// TIA Portal V16 export
// export: Created 2024-12-03T15:41:42.3875884Z, ExportSetting WithDefaults, DisplayName Totally Integrated Automation Portal, DisplayVersion V16 Update 6, DisplayName TIA Portal Version Control Interface, DisplayVersion V16 Update 2, DisplayName TIA Portal Openness, DisplayVersion V16 Update 6, DisplayName TIA Portal Teamcenter Gateway, DisplayVersion V16, DisplayName SINAMICS Startdrive Advanced, DisplayVersion V16 Update 5, DisplayName SINAMICS Startdrive G130, G150, S120, S150, SINAMICS MV, S210, DisplayVersion V16 Update 5, DisplayName SINAMICS Startdrive G110M, G120, G120C, G120D, G120P, G115D, DisplayVersion V16 Update 5, DisplayName STEP 7 Professional, DisplayVersion V16 Update 6, DisplayName STEP 7 Safety, DisplayVersion V16, DisplayName WinCC Advanced / Unified PC, DisplayVersion V16 Update 6
FUNCTION_BLOCK "LC_Cognex_DataMan_FB"   // FB15, SCL
{ S7_Optimized_Access := 'TRUE' }
VERSION : 0.1
// stored: AutoNumber true, IsIECCheckEnabled false, IsRetainMemResEnabled false, MemoryReserve 100, SetENOAutomatically false, UDAEnableTagReadback false
   VAR_OUTPUT
      O_Tracking : "Tracking_Simple_UDT_1";
      O_NewResult : Bool;
   END_VAR
   VAR_IN_OUT
      IO_BarcodeScanner : "COGNEX_DATAMAN_LOGIC_UDT";
      IO_UpstreamConv : "Conveyor_UDT";
      IO_CurrentStream : "Conveyor_UDT";
   END_VAR
   VAR
      measureBoxTimer : TONR_TIME;
      scanTimer { S7_SetPoint := 'True'} : TONR_TIME;
      boxLength { S7_SetPoint := 'True'} : Time;
      stepNumber : DInt;
      Step_10_WaitForTrigger : "StepperController";
      Step_20_OnDelay { S7_SetPoint := 'True'} : "StepperController";
      Step_30_Scan { S7_SetPoint := 'True'} : "StepperController";
      Step_40_ParseResult { S7_SetPoint := 'True'} : "StepperController";
      Step_50_ParcelsToClose { S7_SetPoint := 'True'} : "StepperController";
   END_VAR
   VAR_TEMP
      T_Condition : Bool;
      T_Dummy : Bool;
   END_VAR
BEGIN
   REGION #init

       IF #stepNumber = 0 THEN
           #stepNumber := 10;
       END_IF;

   END_REGION

   REGION Measure box

       #measureBoxTimer(IN := #IO_UpstreamConv.Input.SensorAtEndLogic.State
                        AND #IO_UpstreamConv.Input.Running_FB,
                        PT := T#10s);

       IF #IO_UpstreamConv.Input.SensorAtEndLogic.State THEN
           #boxLength := #measureBoxTimer.ET;
           PRESET_TIMER(PT:= #boxLength + #IO_BarcodeScanner.Settings.OffDelay, "TIMER" := #scanTimer);
       END_IF;

       IF NOT #IO_UpstreamConv.Input.SensorAtEndLogic.State THEN
           RESET_TIMER(#measureBoxTimer);
       END_IF;

   END_REGION

   REGION STEP  10: Standby wait FOR trigger

       #T_Condition :=
       #IO_UpstreamConv.Input.SensorAtEndLogic.State
       AND #IO_UpstreamConv.Input.Running_FB
       AND #IO_UpstreamConv.Cmd.ReadyToSent
       AND #IO_CurrentStream.Cmd.ReadyToReceive;

       #Step_10_WaitForTrigger(I_StepNumber := 10,
                               I_NextStepNumber := 20,
                               I_ErrorStepNumber := 50,
                               I_Condition := #T_Condition AND #IO_BarcodeScanner.Status.ReadyForNewScan,
                               I_ErrorConditon := #T_Condition AND NOT #IO_BarcodeScanner.Status.ReadyForNewScan,
                               I_ConditionTIme := T#0ms,
                               I_IgnoreTimeOut := TRUE,
                               IO_StepNumber := #stepNumber);

       IF #Step_10_WaitForTrigger.O_ConditionTrans
           OR #Step_10_WaitForTrigger.O_ErrorTrans THEN
           #IO_BarcodeScanner.Tracking.ID := #IO_UpstreamConv.TrackingStat.Current.ID;
       END_IF;

   END_REGION

   REGION STEP 20: Start trigger command on delay

       #T_Condition := TRUE;

       #Step_20_OnDelay(I_StepNumber := 20,
                               I_NextStepNumber := 30,
                               I_Condition := #T_Condition,
                               I_ConditionTIme := #IO_BarcodeScanner.Settings.OnDelay,
                               I_PauseTimeOut := NOT #IO_CurrentStream.Input.Running_FB,
                               I_AccumulateConditionTIme := TRUE,
                               I_IgnoreTimeOut := TRUE,
                               IO_StepNumber := #stepNumber);

   END_REGION

   REGION STEP 30: TRIGGER MEASURE TIME + OFF DELAY

       //Timer must be external
       #scanTimer(IN:=#stepNumber = 30 AND ( #IO_CurrentStream.Input.Running_FB OR #IO_CurrentStream.Input.SensorAtEndLogic.State),
                  R:=#stepNumber <> 30,
                  Q=> #T_Dummy,
                  PT:=#boxLength);

       #T_Condition := #scanTimer.Q;

       #Step_30_Scan(I_StepNumber := 30,
                               I_NextStepNumber := 40,
                               I_Condition := #T_Condition,
                               I_ConditionTIme := T#0ms,
                               I_IgnoreTimeOut := TRUE,
                               IO_StepNumber := #stepNumber);

   END_REGION

   REGION STEP40: Wait for result

       #Step_40_ParseResult(I_StepNumber:=40,
                            I_NextStepNumber:=10,
                            I_TimeOutStepNumber:=10,
                            I_ConditionTIme := t#0s,
                            I_Condition:=#IO_BarcodeScanner.ReadingResult.NewResult_Pulse,
                            I_TimeOutTime:=#IO_BarcodeScanner.Settings.TimeOut,
                            IO_StepNumber:=#stepNumber);

       IF #IO_BarcodeScanner.ReadingResult.NewResult_Pulse THEN
           "Test_DB".Counter += 1;
       END_IF;

   END_REGION

   REGION STPEP 50: Parcels to close

       #Step_50_ParcelsToClose(I_StepNumber := 50,
                            I_NextStepNumber := 10,
                            I_TimeOutStepNumber := 10,
                            I_Condition := NOT #IO_CurrentStream.Input.SensorAtStartLogic.State,
                            I_IgnoreTimeOut := true,
                            I_TimeOutTime := #IO_BarcodeScanner.Settings.TimeOut,
                            IO_StepNumber := #stepNumber);

   END_REGION

   REGION Scanner commands

       #IO_BarcodeScanner.Cmd.ScanAuto := #stepNumber = 30;

   END_REGION

   REGION OUTPUTS

       #O_Tracking := "Tracking_DB".EmptyTrackingSimple;
       #O_NewResult := FALSE;

       IF #Step_40_ParseResult.O_ConditionTrans THEN
           #O_Tracking.ID := #IO_BarcodeScanner.Tracking.ID;
           #O_Tracking.Barcode := #IO_BarcodeScanner.ReadingResult.Barcode_Pulse;
           #O_Tracking.GoodRead := #IO_BarcodeScanner.ReadingResult.GoodRead_Pulse;
           #O_NewResult := true;
       END_IF;

       IF #Step_50_ParcelsToClose.O_ConditionTrans THEN
           #O_Tracking.ID := #IO_BarcodeScanner.Tracking.ID;
           #O_Tracking.Barcode:= 'Parcels TO close';
           #O_Tracking.GoodRead := #IO_BarcodeScanner.ReadingResult.GoodRead_Pulse;
           #O_NewResult := true;
       END_IF;

   END_REGION
END_FUNCTION_BLOCK
